// TIA Portal V16 export
// export: Created 2024-12-03T15:41:40.2556272Z, ExportSetting WithDefaults, DisplayName Totally Integrated Automation Portal, DisplayVersion V16 Update 6, DisplayName TIA Portal Version Control Interface, DisplayVersion V16 Update 2, DisplayName TIA Portal Openness, DisplayVersion V16 Update 6, DisplayName TIA Portal Teamcenter Gateway, DisplayVersion V16, DisplayName SINAMICS Startdrive Advanced, DisplayVersion V16 Update 5, DisplayName SINAMICS Startdrive G130, G150, S120, S150, SINAMICS MV, S210, DisplayVersion V16 Update 5, DisplayName SINAMICS Startdrive G110M, G120, G120C, G120D, G120P, G115D, DisplayVersion V16 Update 5, DisplayName STEP 7 Professional, DisplayVersion V16 Update 6, DisplayName STEP 7 Safety, DisplayVersion V16, DisplayName WinCC Advanced / Unified PC, DisplayVersion V16 Update 6
FUNCTION_BLOCK "Z_100_LOGIC_FB"   // FB19, SCL
{ S7_Optimized_Access := 'TRUE' }
VERSION : 0.1
// stored: AutoNumber true, IsIECCheckEnabled false, IsRetainMemResEnabled false, MemoryReserve 100, SetENOAutomatically false, UDAEnableTagReadback false
   VAR
      CONV_101 : "ZPA_Controller";
      CONV_102L : "ZPA_Controller";
      CONV_102R : "ZPA_Controller";
      CONV_103L : "ZPA_Controller";
      CONV_103R : "ZPA_Controller";
      CONV_104L : "ZPA_Controller";
      CONV_104R : "ZPA_Controller";
      CONV_105L : "ZPA_Controller";
      CONV_105R : "ZPA_Controller";
      CONV_106R : "ZPA_Controller";
      CONV_107R : "ZPA_Controller";
      CONV_108L : "ZPA_Controller";
      CONV_108R : "ZPA_Controller";
      CONV_109L : "ZPA_Controller";
      CONV_109R : "ZPA_Controller";
      CONV_110L : "ZPA_Controller";
      CONV_110R : "ZPA_Controller";
      CONV_111L : "ZPA_Controller";
      CONV_111R : "Intersection_Controller_FB";
      CONV_112R : "ZPA_Controller";
      CONV_113L : "ZPA_Controller";
      CONV_113R : "ZPA_Controller";
      CONV_114L : "ZPA_Controller";
      CONV_114R : "ZPA_Controller";
      CONV_115L : "ZPA_Controller";
      CONV_115R : "ZPA_Controller";
      CONV_202L : "ZPA_Controller";
      CONV_202R : "ZPA_Controller";
      CONV_203L : "ZPA_Controller";
      CONV_203R : "ZPA_Controller";
      CONV_301R : "ZPA_Controller";
      CONV_302L : "ZPA_Controller";
      CONV_302R : "ZPA_Controller";
      CONV_303L : "ZPA_Controller";
      CONV_303R : "ZPA_Controller";
      CONV_304L : "Intersection_Controller_FB";
      CONV_304R : "ZPA_Controller";
      CONV_305R : "ZPA_Controller";
      CONV_107_T_splitter { S7_SetPoint := 'True'} : "TrafficController_INTERSECT_SENDING_FB";
      CONV_112L_T_receive { S7_SetPoint := 'True'} : "TrafficController_INTERSECT_RECEIVE_FB";
   END_VAR
   VAR_TEMP
      T_upstream : "Conveyor_UDT";
      T_Condition : Bool;
   END_VAR
BEGIN
   REGION ROUTER

       "ROUTER_CONV_107_FC"(IO_CONV := "CONV_DB".CONV_106R);

   END_REGION

   REGION TRAFFIC CONTROLLER

       REGION C107

           #CONV_107_T_splitter.I_Option_1_Settings.DownstreamIndex := "West";
           #CONV_107_T_splitter.I_Option_2_Settings.DownstreamIndex := "South";

           #CONV_107_T_splitter(I_Option:="CONV_DB".CONV_106R.TrackingStat.InSending.PLC_Dest,
                                IO_SendingConveyor := "CONV_DB".CONV_106R,
                                IO_IntersectionSettings := "Intersection_DB".C107);

       END_REGION

       REGION C112

           #CONV_112L_T_receive(I_IntersectionConveyor:="CONV_DB".CONV_113L,
                                IO_IntersectionSettings:="Intersection_DB".C113L,
                                IO_SendingConveyor_1:="CONV_DB".CONV_113L,
                                IO_SendingConveyor_2:="CONV_DB".CONV_305R);

       END_REGION

   END_REGION

   REGION MAIN LOOP

       REGION CONV_101

           #CONV_101(
                     IO_Upstream := "CONV_DB".CONV_115L,
                     IO_DownStream := "CONV_DB".CONV_102L,
                     IO_COnv := "CONV_DB".CONV_101);

       END_REGION

       REGION CONV_102L

           #CONV_102L(
                      IO_Upstream := "CONV_DB".CONV_101,
                      IO_DownStream := "CONV_DB".CONV_102R,
                      IO_COnv := "CONV_DB".CONV_102L);

       END_REGION

       REGION CONV_102R

           #CONV_102R(
                      IO_Upstream := "CONV_DB".CONV_102L,
                      IO_DownStream := "CONV_DB".CONV_103L,
                      IO_COnv := "CONV_DB".CONV_102R);

       END_REGION

       REGION CONV_103L

           #CONV_103L(
                      IO_Upstream := "CONV_DB".CONV_102R,
                      IO_DownStream := "CONV_DB".CONV_103R,
                      IO_COnv := "CONV_DB".CONV_103L);

       END_REGION

       REGION CONV_103R

           #CONV_103R(
                      IO_Upstream := "CONV_DB".CONV_103L,
                      IO_DownStream := "CONV_DB".CONV_104R,
                      IO_COnv := "CONV_DB".CONV_103R);

       END_REGION

       REGION CONV_104R

           #CONV_104R(
                      IO_Upstream := "CONV_DB".CONV_103R,
                      IO_DownStream := "CONV_DB".CONV_104L,
                      IO_COnv := "CONV_DB".CONV_104R);

       END_REGION

       REGION CONV_104L

           #CONV_104L(
                      IO_Upstream := "CONV_DB".CONV_104R,
                      IO_DownStream := "CONV_DB".CONV_105R,
                      IO_COnv := "CONV_DB".CONV_104L);

       END_REGION

       REGION CONV_105R

           #CONV_105R(
                      IO_Upstream := "CONV_DB".CONV_104L,
                      IO_DownStream := "CONV_DB".CONV_105L,
                      IO_COnv := "CONV_DB".CONV_105R);

       END_REGION

       REGION CONV_105L

           #CONV_105L(
                      IO_Upstream := "CONV_DB".CONV_105R,
                      IO_DownStream := "CONV_DB".CONV_106R,
                      IO_COnv := "CONV_DB".CONV_105L);

       END_REGION

       REGION CONV_106R SCANNER

           "SCAN_100"(IO_Upstream:="CONV_DB".CONV_105L,
                      IO_CurrentStream:="CONV_DB".CONV_106R,
                      IO_Scanner_1:="Scanners_DB".SCAN_100);

           #CONV_106R(
                      IO_Upstream := "CONV_DB".CONV_105L,
                      IO_DownStream := "CONV_DB".CONV_107R,
                      IO_COnv := "CONV_DB".CONV_106R);

       END_REGION

       REGION CONV_107R DIVERTER

           REGION DIVERTER CONTROLLER

               IF "Intersection_DB".C107.DownstreamIndex = "West" THEN
                   "MOT_CLX_DB".MOT_107L.Cmd.SetPointDegAuto :=
                   "MOT_CLX_DB".MOT_107L.Settings.Option_1;
               END_IF;

               IF "Intersection_DB".C107.DownstreamIndex = "South" THEN
                   "MOT_CLX_DB".MOT_107L.Cmd.SetPointDegAuto :=
                   "MOT_CLX_DB".MOT_107L.Settings.Option_2;
               END_IF;

           END_REGION

           #CONV_107R(
                      IO_Upstream := "CONV_DB".CONV_106R,
                      IO_DownStream := "CONV_DB".CONV_108R,
                      IO_COnv := "CONV_DB".CONV_107R);

       END_REGION

       REGION CONV_108R

           #CONV_108R(I_ConnectUpStream := "Intersection_DB".C107.DownstreamIndex = "West",
                      IO_Upstream := "CONV_DB".CONV_107R,
                      IO_DownStream := "CONV_DB".CONV_108L,
                      IO_COnv := "CONV_DB".CONV_108R);

       END_REGION

       REGION CONV_108L

           #CONV_108L(
                      IO_Upstream := "CONV_DB".CONV_108R,
                      IO_DownStream := "CONV_DB".CONV_109R,
                      IO_COnv := "CONV_DB".CONV_108L);

       END_REGION

       REGION CONV_109R

           #CONV_109R(
                      IO_Upstream := "CONV_DB".CONV_108L,
                      IO_DownStream := "CONV_DB".CONV_109L,
                      IO_COnv := "CONV_DB".CONV_109R);

       END_REGION

       REGION CONV_109L

           #CONV_109L(
                      IO_Upstream := "CONV_DB".CONV_109R,
                      IO_DownStream := "CONV_DB".CONV_110R,
                      IO_COnv := "CONV_DB".CONV_109L);

       END_REGION

       REGION CONV_110R

           #CONV_110R(
                      IO_Upstream := "CONV_DB".CONV_109L,
                      IO_DownStream := "CONV_DB".CONV_110L,
                      IO_COnv := "CONV_DB".CONV_110R);

       END_REGION

       REGION CONV_110L

           #CONV_110L(
                      IO_Upstream := "CONV_DB".CONV_110R,
                      IO_DownStream := "CONV_DB".CONV_111R,
                      IO_COnv := "CONV_DB".CONV_110L);

       END_REGION

       REGION CONV_111R INTERSECTION

           #CONV_111R(
                      I_Conv_North := "CONV_DB".empty,
                      I_Conv_East := "CONV_DB".CONV_110L,
                      I_Conv_South := "CONV_DB".CONV_203R_BELTS,
                      I_Conv_West := "CONV_DB".CONV_111L,
                      I_Settings := "Intersection_DB".C111R,
                      IO_Conv_1 := "CONV_DB".CONV_111R,
                      IO_Conv_2 := "CONV_DB".CONV_201R_BELTS,
                      IO_Transfer := "TRANSFER_DB".T201L);


       END_REGION

       REGION CONV_111L

           #CONV_111L(
                      IO_Upstream := "CONV_DB".CONV_111R,
                      IO_DownStream := "CONV_DB".CONV_112R,
                      IO_COnv := "CONV_DB".CONV_111L);

       END_REGION

       REGION CONV_112R

           #CONV_112R(
                      IO_Upstream := "CONV_DB".CONV_111L,
                      IO_DownStream := "CONV_DB".CONV_113L,
                      IO_COnv := "CONV_DB".CONV_112R);

       END_REGION

       REGION CONV_113L

           #CONV_113L(
                      IO_Upstream := "CONV_DB".CONV_112R,
                      IO_DownStream := "CONV_DB".CONV_114R,
                      IO_COnv := "CONV_DB".CONV_113L);

       END_REGION

       REGION CONV_114R

           #CONV_114R(
                      IO_Upstream := "CONV_DB".CONV_113L,
                      IO_DownStream := "CONV_DB".CONV_114L,
                      IO_COnv := "CONV_DB".CONV_114R);

       END_REGION

       REGION CONV_114L

           #CONV_114L(
                      IO_Upstream := "CONV_DB".CONV_114R,
                      IO_DownStream := "CONV_DB".CONV_115R,
                      IO_COnv := "CONV_DB".CONV_114L);

       END_REGION

       REGION CONV_115R

           #CONV_115R(
                      IO_Upstream := "CONV_DB".CONV_114L,
                      IO_DownStream := "CONV_DB".CONV_115L,
                      IO_COnv := "CONV_DB".CONV_115R);

       END_REGION

       REGION CONV_115L

           #CONV_115L(
                      IO_Upstream := "CONV_DB".CONV_115R,
                      IO_DownStream := "CONV_DB".CONV_101,
                      IO_COnv := "CONV_DB".CONV_115L);

       END_REGION


   END_REGION

   REGION SIDE LANE

       REGION CONV_301R

           #CONV_301R(I_ConnectUpStream := "Intersection_DB".C107.DownstreamIndex = "South",
                      IO_Upstream := "CONV_DB".CONV_107R,
                      IO_DownStream := "CONV_DB".CONV_302L,
                      IO_COnv := "CONV_DB".CONV_301R);


       END_REGION

       REGION CONV_302L

           #CONV_302L(
                      IO_Upstream := "CONV_DB".CONV_301R,
                      IO_DownStream := "CONV_DB".CONV_302R,
                      IO_COnv := "CONV_DB".CONV_302L);

       END_REGION

       REGION CONV_302R

           #CONV_302R(
                      IO_Upstream := "CONV_DB".CONV_302L,
                      IO_DownStream := "CONV_DB".CONV_303L,
                      IO_COnv := "CONV_DB".CONV_302R);

       END_REGION

       REGION CONV_303L

           #CONV_303L(
                      IO_Upstream := "CONV_DB".CONV_302R,
                      IO_DownStream := "CONV_DB".CONV_303R,
                      IO_COnv := "CONV_DB".CONV_303L);

       END_REGION

       REGION CONV_303R

           #CONV_303R(
                      IO_Upstream := "CONV_DB".CONV_303L,
                      IO_DownStream := "CONV_DB".CONV_304L,
                      IO_COnv := "CONV_DB".CONV_303R);

       END_REGION

       REGION CONV_304L

           #CONV_304L(
                      I_Conv_North := "CONV_DB".CONV_201R_BELTS,
                      I_Conv_East := "CONV_DB".CONV_303R,
                      I_Conv_South := "CONV_DB".empty,
                      I_Conv_West := "CONV_DB".CONV_304R,
                      I_Settings := "Intersection_DB".C304L,
                      IO_Conv_1 := "CONV_DB".CONV_304L,
                      IO_Conv_2 := "CONV_DB".CONV_203R_BELTS,
                      IO_Transfer := "TRANSFER_DB".T203L);


       END_REGION

       REGION CONV_304R

           #CONV_304R(
                      IO_Upstream := "CONV_DB".CONV_304L,
                      IO_DownStream := "CONV_DB".CONV_305R,
                      IO_COnv := "CONV_DB".CONV_304R);

       END_REGION

       REGION CONV_305R

           #CONV_305R(
                      IO_Upstream := "CONV_DB".CONV_304R,
                      IO_DownStream := "CONV_DB".CONV_112R,
                      IO_COnv := "CONV_DB".CONV_305R);

       END_REGION

   END_REGION
END_FUNCTION_BLOCK
